FUNCTION_BLOCK Cata (* Service Interface Function Block Type *)
  (* Standard: 61499-1 Annex A; Description: Copyright (c) 2017 fortiss GmbH This program and the accompanying materials are made available under the terms of the Eclipse Public License 2.0 which is available at https://www.eclipse.org/legal/epl-2.0/ SPDX-License-Identifier: EPL-2.0 *)
  (* Version 1.0, 2017-09-21, Alois Zoitl, fortiss GmbH, initial API and implementation and/or initial documentation *)
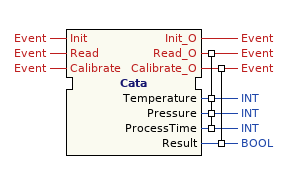
  EVENT_INPUT
    Init;
    Read;
    Calibrate; {SET_ATTRIBUTE(OpcUa, Method)}
  END_EVENT
  EVENT_OUTPUT
    Init_O;
    Read_O WITH Temperature, Pressure, ProcessTime;
    Calibrate_O WITH Result;
  END_EVENT
  VAR_OUTPUT
    Temperature : INT; {SET_ATTRIBUTE(OpcUa, Variable)}
    Pressure : INT; {SET_ATTRIBUTE(OpcUa, Variable)}
    ProcessTime : INT; {SET_ATTRIBUTE(OpcUa, Variable)}
    Result : BOOL; {SET_ATTRIBUTE(OpcUa, Calibrate)}
  END_VAR
END_FUNCTION_BLOCK
(* other elements stored in the file *)
(* SelfDiscription FBType=DEVICE.SENSOR *)
